// TIA Portal V18 export
FUNCTION_BLOCK "ST10_Flow2_A1TableUnloading"   // FB1072, GRAPH
// stored: AcknowledgeErrorsRequired false, AutoNumber false, GraphVersion 6.0, InitialValuesAcquisition false, SetENOAutomatically false
   // inherited from GRAPH_BASE
   VAR_INPUT
      iSysInface : "RCS_SysComInterface_V1";
   END_VAR
   VAR_IN_OUT
      ioPM_Inface : "RCS_PMInterface_V1";
      ioStatus : Int;
   END_VAR
   VAR
      sCtrlMode { S7_SetPoint := 'True'} : "SysFlowCtrlGraph";
      sUpdMES_Data : Bool;   // 更新MES数据
      工件放行中 : Bool;
      前站站号 { ExternalAccessible := 'False'; ExternalVisible := 'False'; ExternalWritable := 'False'} : UInt;
      本站站号 { ExternalAccessible := 'False'; ExternalVisible := 'False'; ExternalWritable := 'False'} : UInt;
      弹窗Temp : Array[1..10] of Int;
      AlarmID : Int;
      TON { S7_SetPoint := 'True'} : Array[0..10] of TON_TIME;
      TOF { S7_SetPoint := 'True'} : Array[0..10] of TOF_TIME;
      sUP { S7_SetPoint := 'True'} : Array[0..10] of Bool;
      更新RFID完成 : Bool;
   END_VAR
   VAR_TEMP
      Tempresult : USInt;
      本站站号乘10 : UInt;
   END_VAR
   // // TON[0] : 托盘流入1托盘到位传感器 / iA-Rotating product Check
   // // TON[1] : 托盘流入1托盘到位传感器
   // // TON[2] : 托盘流入1产品有无传感器
   // // TON[3] : 托盘流入1产品有无传感器
   // // TON[4] : 托盘流入1姿态检测光电2
   // // TON[5] : 托盘流入1姿态检测光电3
   // // TON[0].Q : 托盘流入1托盘到位 / iA-Rotating product Check
   // // TON[1].Q : 托盘流入1托盘无
   // // TON[2].Q : 托盘流入1有产品
   // // TON[3].Q : 托盘流入1无产品
   // // TON[4].Q : 托盘流入1姿态检测光电2
   // // TON[5].Q : 托盘流入1姿态检测光电3
   // // TOF[1] : iA-Rotating product Check
BEGIN
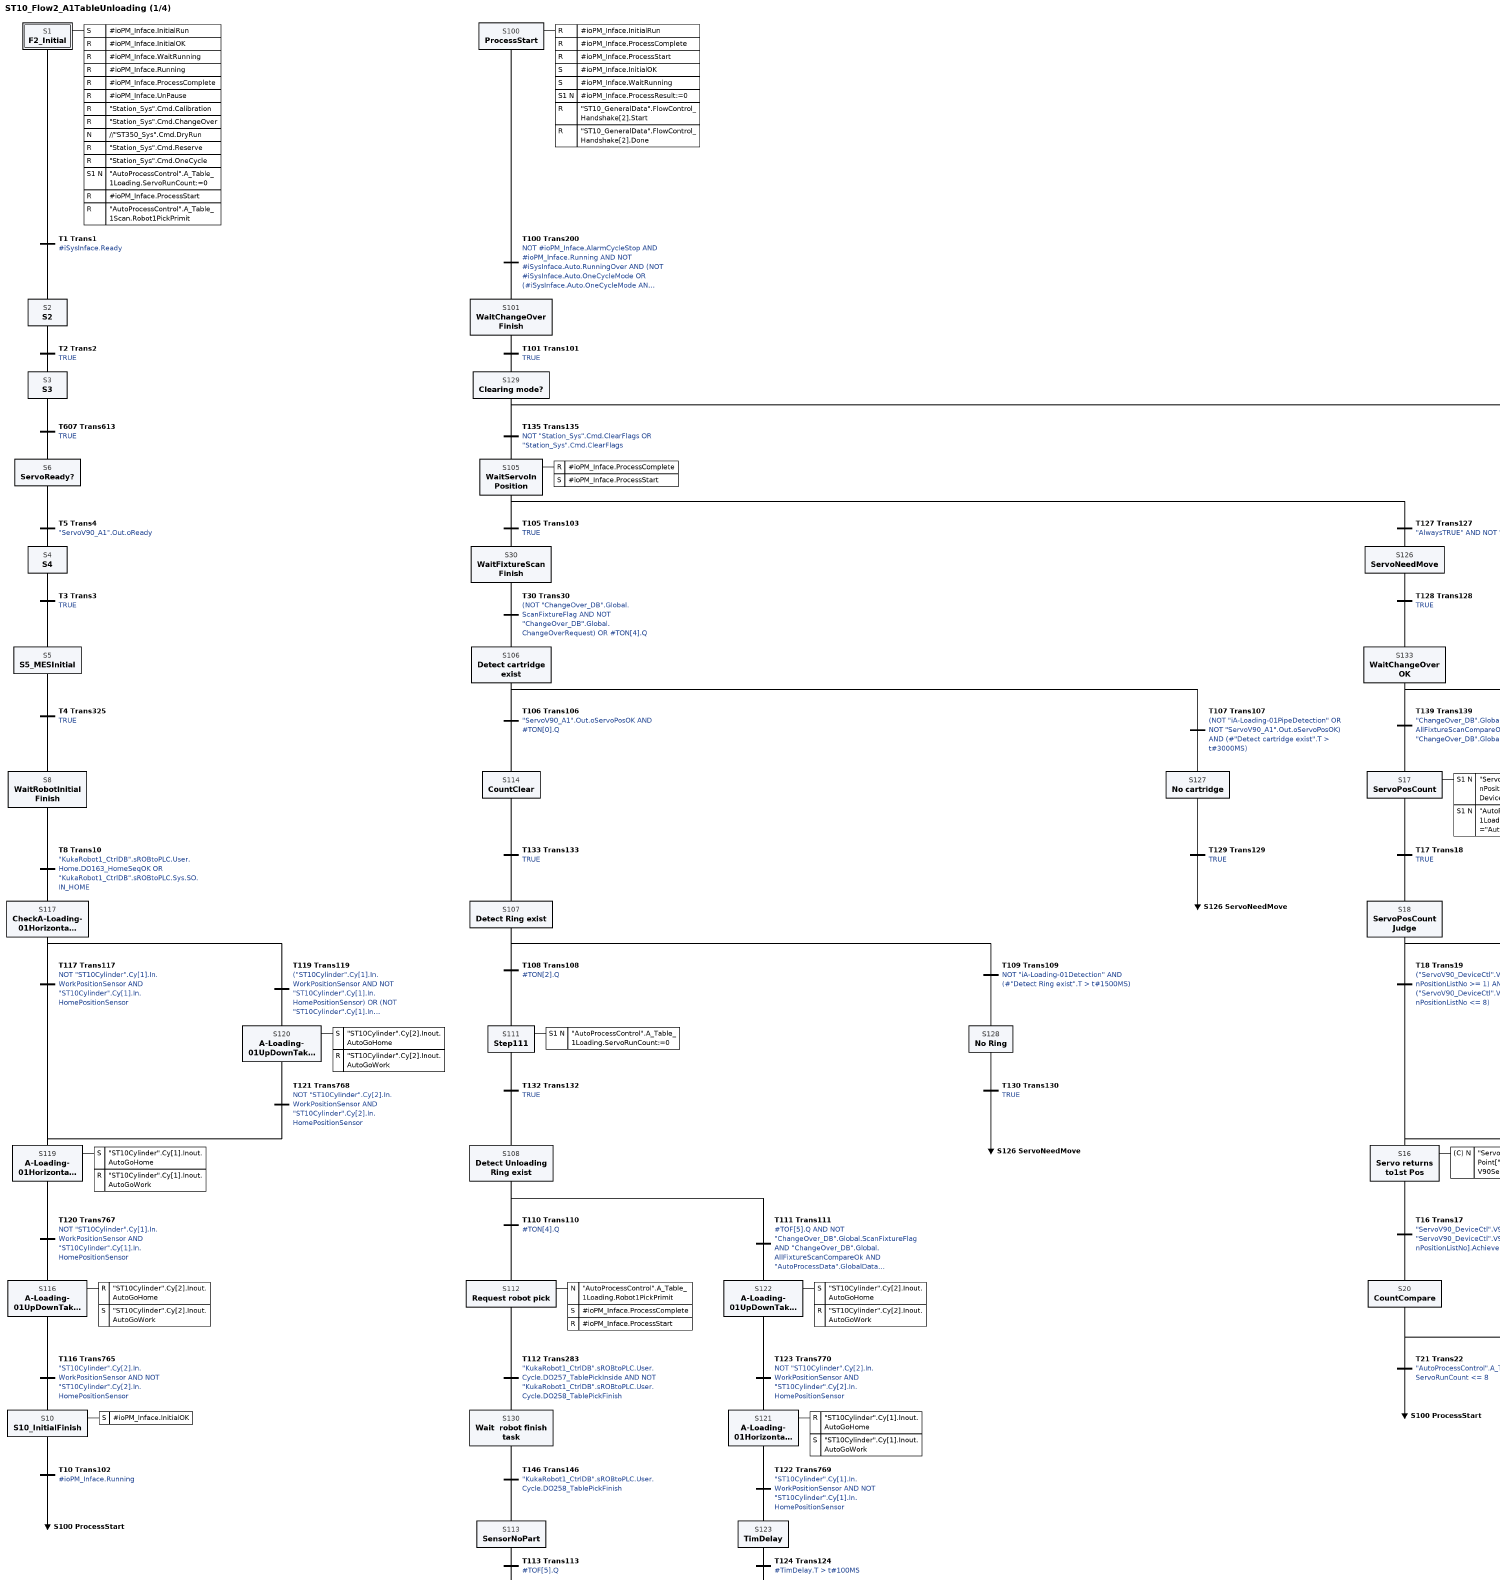
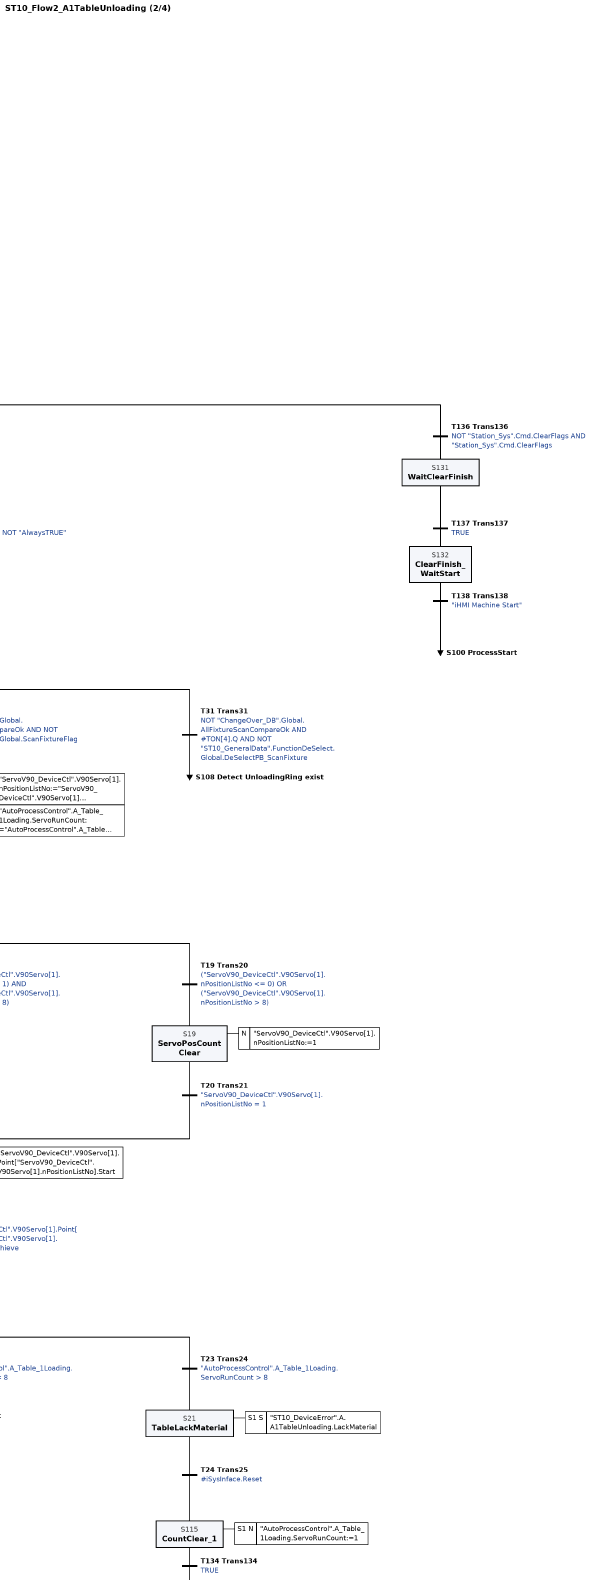
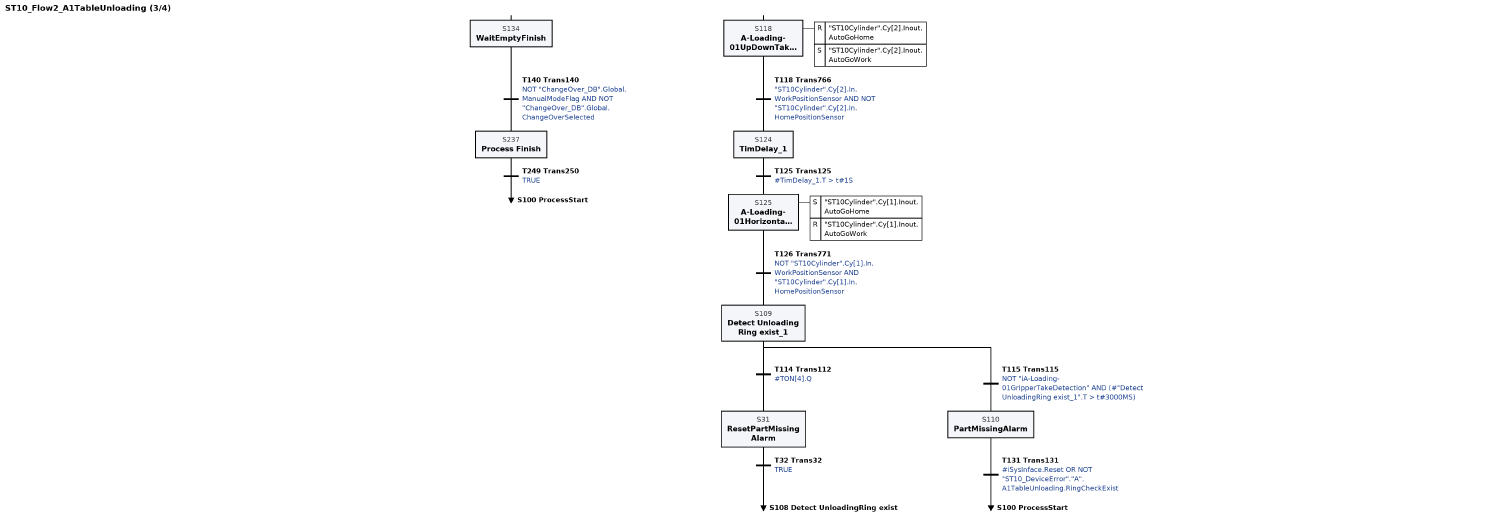
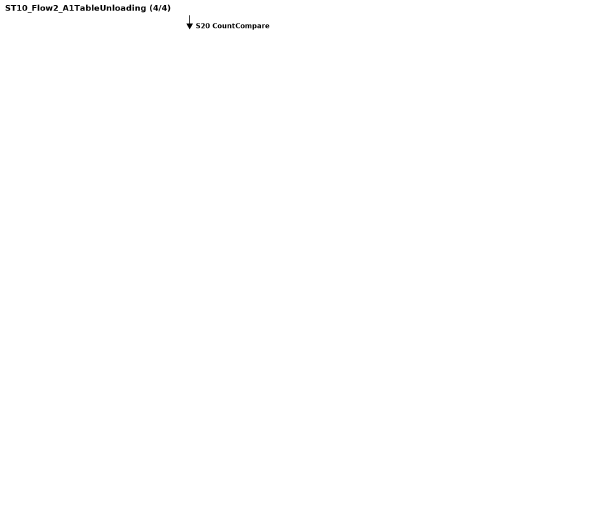
   // permanent pre-instructions
   NETWORK 1
      #TON[10].TON(IN := "AlwaysTRUE" AND "Station_Sys".Alarm.ImmediatelyStop, PT := T#300ms);
      #ioPM_Inface.AlarmImdilyStop := #TON[10].Q;
      #ioPM_Inface.AlarmCycleStop := "AlwaysTRUE" AND "Station_Sys".Alarm.CycleStop;
   NETWORK 2
      IF NOT False THEN
          #sCtrlMode(iSysInface := #iSysInface, ioPM_Inface := #ioPM_Inface, ioGraphCtrl := #RT_DATA.MOP);   // "SysFlowCtrlGraph"
      END_IF;
   NETWORK 3
      #TON[0].TON(IN := "AlwaysTRUE" AND "iA-Loading-01PipeDetection", PT := t#500ms);   // 工位11有托盘
      #TOF[1].TOF(IN := "AlwaysTRUE" AND NOT "iA-Loading-01PipeDetection", PT := T#300ms);   // 工位无托盘
      #TON[2].TON(IN := "AlwaysTRUE" AND "iA-Loading-01Detection", PT := T#300ms);
      #TOF[3].TOF(IN := "AlwaysTRUE" AND NOT "iA-Loading-01Detection", PT := T#300ms);
      #TON[4].TON(IN := "AlwaysTRUE" AND "iA-Loading-01GripperTakeDetection", PT := T#300ms);
      #TOF[5].TOF(IN := "AlwaysTRUE" AND NOT "iA-Loading-01GripperTakeDetection", PT := T#300ms);
   NETWORK 4
      #前站站号 := 345;
      #本站站号 := 350;

   // sequencer 1: S01-S99 初始化 / S01-S99 Initial
   INITIAL_STEP F2_Initial:   // S1, max time T#10S, warning time T#7S
              S    #ioPM_Inface.InitialRun
              R    #ioPM_Inface.InitialOK
              R    #ioPM_Inface.WaitRunning
              R    #ioPM_Inface.Running
              R    #ioPM_Inface.ProcessComplete
              R    #ioPM_Inface.UnPause
              R    "Station_Sys".Cmd.Calibration
              R    "Station_Sys".Cmd.ChangeOver
                   //"ST350_Sys".Cmd.DryRun
              R    "Station_Sys".Cmd.Reserve
              R    "Station_Sys".Cmd.OneCycle
          S1  N    "AutoProcessControl".A_Table_1Loading.ServoRunCount:=0
              R    #ioPM_Inface.ProcessStart
              R    "AutoProcessControl".A_Table_1Scan.Robot1PickPrimit
              R    "AutoProcessControl".A_Table_1Loading.Robot1PickPrimit
              R    "AutoProcessControl".A_Table_2Scan.Robot3PickPrimit
              R    "AutoProcessControl".A_Table_2Loading.Robot3PickPrimit
              R    "AutoProcessControl".A_ScanRotary.Robot1PickPrimit
              R    "AutoProcessControl".A_ScanRotary.Robot1PutPrimit
              R    "AutoProcessControl".H_ShafeLine.Robot1PickPrimit
              R    "AutoProcessControl".J_MagnetLine.Robot2PickPrimit
              R    "AutoProcessControl".K_ShafeLine.Robot2PickPrimit
              R    "AutoProcessControl".L_ShafeLine.Robot3PutPrimit
   END_STEP
   TRANSITION Trans1 FROM F2_Initial TO S2   // T1
      := #iSysInface.Ready;
   END_TRANSITION
   STEP S2:   // S2, max time T#10S, warning time T#7S
   END_STEP
   TRANSITION Trans2 FROM S2 TO S3   // T2
      := TRUE;
   END_TRANSITION
   STEP S4:   // S4, max time T#10S, warning time T#7S
   END_STEP
   TRANSITION Trans3 FROM S4 TO S5_MESInitial   // T3
      := TRUE;
   END_TRANSITION
   STEP S5_MESInitial:   // S5, max time T#10S, warning time T#7S
   END_STEP
   TRANSITION Trans325 FROM S5_MESInitial TO WaitRobotInitialFinish   // T4
      := TRUE;
   END_TRANSITION
   STEP S10_InitialFinish:   // S10, max time T#10S, warning time T#7S
              S    #ioPM_Inface.InitialOK
   END_STEP
   TRANSITION Trans102 FROM S10_InitialFinish TO ProcessStart   // T10, jump
      := #ioPM_Inface.Running;
   END_TRANSITION
   STEP S3:   // S3, max time T#10S, warning time T#7S
   END_STEP
   TRANSITION Trans613 FROM S3 TO "ServoReady?"   // T607
      := TRUE;
   END_TRANSITION
   STEP WaitRobotInitialFinish:   // S8, max time T#10S, warning time T#7S
   END_STEP
   TRANSITION Trans10 FROM WaitRobotInitialFinish TO "CheckA-Loading-01HorizontalCylindePos"   // T8
      := "KukaRobot1_CtrlDB".sROBtoPLC.User.Home.DO163_HomeSeqOK OR "KukaRobot1_CtrlDB".sROBtoPLC.Sys.SO.IN_HOME;
   END_TRANSITION
   STEP "A-Loading-01UpDownTakeCylinderToHP_2":   // S120, max time T#10S, warning time T#7S
              S    "ST10Cylinder".Cy[2].Inout.AutoGoHome
              R    "ST10Cylinder".Cy[2].Inout.AutoGoWork
   END_STEP
   TRANSITION Trans768 FROM "A-Loading-01UpDownTakeCylinderToHP_2" TO "A-Loading-01HorizontalCylinderToHP"   // T121
      := NOT "ST10Cylinder".Cy[2].In.WorkPositionSensor AND "ST10Cylinder".Cy[2].In.HomePositionSensor;
   END_TRANSITION
   STEP "CheckA-Loading-01HorizontalCylindePos":   // S117, max time T#10S, warning time T#7S
   END_STEP
   TRANSITION Trans117 FROM "CheckA-Loading-01HorizontalCylindePos" TO "A-Loading-01HorizontalCylinderToHP"   // T117
      := NOT "ST10Cylinder".Cy[1].In.WorkPositionSensor AND "ST10Cylinder".Cy[1].In.HomePositionSensor;
   END_TRANSITION
   TRANSITION Trans119 FROM "CheckA-Loading-01HorizontalCylindePos" TO "A-Loading-01UpDownTakeCylinderToHP_2"   // T119
      := ("ST10Cylinder".Cy[1].In.WorkPositionSensor AND NOT "ST10Cylinder".Cy[1].In.HomePositionSensor) OR (NOT "ST10Cylinder".Cy[1].In.WorkPositionSensor AND NOT "ST10Cylinder".Cy[1].In.HomePositionSensor);
   END_TRANSITION
   STEP "A-Loading-01HorizontalCylinderToHP":   // S119, max time T#10S, warning time T#7S
              S    "ST10Cylinder".Cy[1].Inout.AutoGoHome
              R    "ST10Cylinder".Cy[1].Inout.AutoGoWork
   END_STEP
   TRANSITION Trans767 FROM "A-Loading-01HorizontalCylinderToHP" TO "A-Loading-01UpDownTakeCylinderToWP"   // T120
      := NOT "ST10Cylinder".Cy[1].In.WorkPositionSensor AND "ST10Cylinder".Cy[1].In.HomePositionSensor;
   END_TRANSITION
   STEP "A-Loading-01UpDownTakeCylinderToWP":   // S116, max time T#10S, warning time T#7S
              R    "ST10Cylinder".Cy[2].Inout.AutoGoHome
              S    "ST10Cylinder".Cy[2].Inout.AutoGoWork
   END_STEP
   TRANSITION Trans765 FROM "A-Loading-01UpDownTakeCylinderToWP" TO S10_InitialFinish   // T116
      := "ST10Cylinder".Cy[2].In.WorkPositionSensor AND NOT "ST10Cylinder".Cy[2].In.HomePositionSensor;
   END_TRANSITION
   STEP "ServoReady?":   // S6, max time T#10S, warning time T#7S
   END_STEP
   TRANSITION Trans4 FROM "ServoReady?" TO S4   // T5
      := "ServoV90_A1".Out.oReady;
   END_TRANSITION

   // sequencer 2: S100-S199 等待到位 / S100-S199 CheckSysStatus
   STEP "A-Loading-01HorizontalCylinderToWP_1":   // S121, max time T#10S, warning time T#7S
              R    "ST10Cylinder".Cy[1].Inout.AutoGoHome
              S    "ST10Cylinder".Cy[1].Inout.AutoGoWork
   END_STEP
   TRANSITION Trans769 FROM "A-Loading-01HorizontalCylinderToWP_1" TO TimDelay   // T122
      := "ST10Cylinder".Cy[1].In.WorkPositionSensor AND NOT "ST10Cylinder".Cy[1].In.HomePositionSensor;
   END_TRANSITION
   STEP "A-Loading-01UpDownTakeCylinderToHP3":   // S122, max time T#10S, warning time T#7S
              S    "ST10Cylinder".Cy[2].Inout.AutoGoHome
              R    "ST10Cylinder".Cy[2].Inout.AutoGoWork
   END_STEP
   TRANSITION Trans770 FROM "A-Loading-01UpDownTakeCylinderToHP3" TO "A-Loading-01HorizontalCylinderToWP_1"   // T123
      := NOT "ST10Cylinder".Cy[2].In.WorkPositionSensor AND "ST10Cylinder".Cy[2].In.HomePositionSensor;
   END_TRANSITION
   STEP TimDelay:   // S123, max time T#10S, warning time T#7S
   END_STEP
   TRANSITION Trans124 FROM TimDelay TO "A-Loading-01UpDownTakeCylinderToWP_1"   // T124
      := #TimDelay.T > t#100MS;
   END_TRANSITION
   STEP SensorNoPart:   // S113, max time T#10S, warning time T#7S
   END_STEP
   TRANSITION Trans113 FROM SensorNoPart TO WaitEmptyFinish   // T113
      := #TOF[5].Q;
   END_TRANSITION
   STEP ProcessStart:   // S100, max time T#10S, warning time T#7S
      // 自动等待开始运行
              R    #ioPM_Inface.InitialRun
              R    #ioPM_Inface.ProcessComplete
              R    #ioPM_Inface.ProcessStart
              S    #ioPM_Inface.InitialOK
              S    #ioPM_Inface.WaitRunning
          S1  N    #ioPM_Inface.ProcessResult:=0
              R    "ST10_GeneralData".FlowControl_Handshake[2].Start
              R    "ST10_GeneralData".FlowControl_Handshake[2].Done
   END_STEP
   TRANSITION Trans200 FROM ProcessStart TO WaitChangeOverFinish   // T100
      := NOT #ioPM_Inface.AlarmCycleStop AND #ioPM_Inface.Running AND NOT #iSysInface.Auto.RunningOver AND (NOT #iSysInface.Auto.OneCycleMode OR (#iSysInface.Auto.OneCycleMode AND #ioPM_Inface.TriggerOneCycle));
   END_TRANSITION
   STEP TimDelay_1:   // S124, max time T#10S, warning time T#7S
   END_STEP
   TRANSITION Trans125 FROM TimDelay_1 TO "A-Loading-01HorizontalCylinderToHP_1"   // T125
      := #TimDelay_1.T > t#1S;
   END_TRANSITION
   STEP "Process Finish":   // S237, max time T#10S, warning time T#7S
   END_STEP
   TRANSITION Trans250 FROM "Process Finish" TO ProcessStart   // T249, jump
      := TRUE;
   END_TRANSITION
   STEP "A-Loading-01HorizontalCylinderToHP_1":   // S125, max time T#10S, warning time T#7S
              S    "ST10Cylinder".Cy[1].Inout.AutoGoHome
              R    "ST10Cylinder".Cy[1].Inout.AutoGoWork
   END_STEP
   TRANSITION Trans771 FROM "A-Loading-01HorizontalCylinderToHP_1" TO "Detect UnloadingRing exist_1"   // T126
      := NOT "ST10Cylinder".Cy[1].In.WorkPositionSensor AND "ST10Cylinder".Cy[1].In.HomePositionSensor;
   END_TRANSITION
   STEP "No cartridge":   // S127, max time T#10S, warning time T#7S
   END_STEP
   TRANSITION Trans129 FROM "No cartridge" TO ServoNeedMove   // T129, jump
      := TRUE;
   END_TRANSITION
   STEP "A-Loading-01UpDownTakeCylinderToWP_1":   // S118, max time T#10S, warning time T#7S
              R    "ST10Cylinder".Cy[2].Inout.AutoGoHome
              S    "ST10Cylinder".Cy[2].Inout.AutoGoWork
   END_STEP
   TRANSITION Trans766 FROM "A-Loading-01UpDownTakeCylinderToWP_1" TO TimDelay_1   // T118
      := "ST10Cylinder".Cy[2].In.WorkPositionSensor AND NOT "ST10Cylinder".Cy[2].In.HomePositionSensor;
   END_TRANSITION
   STEP ServoNeedMove:   // S126, max time T#10S, warning time T#7S
   END_STEP
   TRANSITION Trans128 FROM ServoNeedMove TO WaitChangeOverOK   // T128
      := TRUE;
   END_TRANSITION
   STEP WaitChangeOverFinish:   // S101, max time T#10S, warning time T#7S
   END_STEP
   TRANSITION Trans101 FROM WaitChangeOverFinish TO "Clearing mode?"   // T101
      := TRUE;
   END_TRANSITION
   STEP WaitServoInPosition:   // S105, max time T#10S, warning time T#7S
              R    #ioPM_Inface.ProcessComplete
              S    #ioPM_Inface.ProcessStart
   END_STEP
   TRANSITION Trans103 FROM WaitServoInPosition TO WaitFixtureScanFinish   // T105
      := TRUE;
   END_TRANSITION
   TRANSITION Trans127 FROM WaitServoInPosition TO ServoNeedMove   // T127
      := "AlwaysTRUE" AND NOT "AlwaysTRUE";
   END_TRANSITION
   STEP "Detect cartridge exist":   // S106, max time T#10S, warning time T#7S
   END_STEP
   TRANSITION Trans106 FROM "Detect cartridge exist" TO CountClear   // T106
      := "ServoV90_A1".Out.oServoPosOK AND #TON[0].Q;
   END_TRANSITION
   TRANSITION Trans107 FROM "Detect cartridge exist" TO "No cartridge"   // T107
      := (NOT "iA-Loading-01PipeDetection" OR NOT "ServoV90_A1".Out.oServoPosOK) AND (#"Detect cartridge exist".T > t#3000MS);
   END_TRANSITION
   STEP "Detect UnloadingRing exist":   // S108, max time T#10S, warning time T#7S
   END_STEP
   TRANSITION Trans110 FROM "Detect UnloadingRing exist" TO "Request robot pick"   // T110
      := #TON[4].Q;
   END_TRANSITION
   TRANSITION Trans111 FROM "Detect UnloadingRing exist" TO "A-Loading-01UpDownTakeCylinderToHP3"   // T111
      := #TOF[5].Q AND NOT "ChangeOver_DB".Global.ScanFixtureFlag AND "ChangeOver_DB".Global.AllFixtureScanCompareOk AND "AutoProcessData".GlobalData.Table1CodeOKFlag;
   END_TRANSITION
   STEP "Detect Ring exist":   // S107, max time T#10S, warning time T#7S
   END_STEP
   TRANSITION Trans108 FROM "Detect Ring exist" TO Step111   // T108
      := #TON[2].Q;
   END_TRANSITION
   TRANSITION Trans109 FROM "Detect Ring exist" TO "No Ring"   // T109
      := NOT "iA-Loading-01Detection" AND (#"Detect Ring exist".T > t#1500MS);
   END_TRANSITION
   STEP "Wait  robot finish task":   // S130, max time T#10S, warning time T#7S
   END_STEP
   TRANSITION Trans146 FROM "Wait  robot finish task" TO SensorNoPart   // T146
      := "KukaRobot1_CtrlDB".sROBtoPLC.User.Cycle.DO258_TablePickFinish;
   END_TRANSITION
   STEP "Request robot pick":   // S112, max time T#10S, warning time T#7S
              N    "AutoProcessControl".A_Table_1Loading.Robot1PickPrimit
              S    #ioPM_Inface.ProcessComplete
              R    #ioPM_Inface.ProcessStart
   END_STEP
   TRANSITION Trans283 FROM "Request robot pick" TO "Wait  robot finish task"   // T112
      := "KukaRobot1_CtrlDB".sROBtoPLC.User.Cycle.DO257_TablePickInside AND NOT "KukaRobot1_CtrlDB".sROBtoPLC.User.Cycle.DO258_TablePickFinish;
   END_TRANSITION
   STEP "No Ring":   // S128, max time T#10S, warning time T#7S
   END_STEP
   TRANSITION Trans130 FROM "No Ring" TO ServoNeedMove   // T130, jump
      := TRUE;
   END_TRANSITION
   STEP "Detect UnloadingRing exist_1":   // S109, max time T#10S, warning time T#7S
   END_STEP
   TRANSITION Trans112 FROM "Detect UnloadingRing exist_1" TO ResetPartMissingAlarm   // T114
      := #TON[4].Q;
   END_TRANSITION
   TRANSITION Trans115 FROM "Detect UnloadingRing exist_1" TO PartMissingAlarm   // T115
      := NOT "iA-Loading-01GripperTakeDetection" AND (#"Detect UnloadingRing exist_1".T > t#3000MS);
   END_TRANSITION
   STEP PartMissingAlarm:   // S110, max time T#10S, warning time T#7S
   END_STEP
   TRANSITION Trans131 FROM PartMissingAlarm TO ProcessStart   // T131, jump
      := #iSysInface.Reset OR NOT "ST10_DeviceError"."A".A1TableUnloading.RingCheckExist;
   END_TRANSITION
   STEP Step111:   // S111, max time T#10S, warning time T#7S
          S1  N    "AutoProcessControl".A_Table_1Loading.ServoRunCount:=0
   END_STEP
   TRANSITION Trans132 FROM Step111 TO "Detect UnloadingRing exist"   // T132
      := TRUE;
   END_TRANSITION
   STEP CountClear:   // S114, max time T#10S, warning time T#7S
   END_STEP
   TRANSITION Trans133 FROM CountClear TO "Detect Ring exist"   // T133
      := TRUE;
   END_TRANSITION
   STEP "Servo returns to1st Pos":   // S16, max time T#10S, warning time T#7S
      interlock C := "ServoV90_A1".Out.oReady;
      (C)     N    "ServoV90_DeviceCtl".V90Servo[1].Point["ServoV90_DeviceCtl".V90Servo[1].nPositionListNo].Start
   END_STEP
   TRANSITION Trans17 FROM "Servo returns to1st Pos" TO CountCompare   // T16
      := "ServoV90_DeviceCtl".V90Servo[1].Point["ServoV90_DeviceCtl".V90Servo[1].nPositionListNo].Achieve;
   END_TRANSITION
   STEP ServoPosCount:   // S17, max time T#10S, warning time T#7S
          S1  N    "ServoV90_DeviceCtl".V90Servo[1].nPositionListNo:="ServoV90_DeviceCtl".V90Servo[1].nPositionListNo+1
          S1  N    "AutoProcessControl".A_Table_1Loading.ServoRunCount:="AutoProcessControl".A_Table_1Loading.ServoRunCount+1
   END_STEP
   TRANSITION Trans18 FROM ServoPosCount TO ServoPosCountJudge   // T17
      := TRUE;
   END_TRANSITION
   STEP ServoPosCountJudge:   // S18, max time T#10S, warning time T#7S
   END_STEP
   TRANSITION Trans19 FROM ServoPosCountJudge TO "Servo returns to1st Pos"   // T18
      := ("ServoV90_DeviceCtl".V90Servo[1].nPositionListNo >= 1) AND ("ServoV90_DeviceCtl".V90Servo[1].nPositionListNo <= 8);
   END_TRANSITION
   TRANSITION Trans20 FROM ServoPosCountJudge TO ServoPosCountClear   // T19
      := ("ServoV90_DeviceCtl".V90Servo[1].nPositionListNo <= 0) OR ("ServoV90_DeviceCtl".V90Servo[1].nPositionListNo > 8);
   END_TRANSITION
   STEP ServoPosCountClear:   // S19, max time T#10S, warning time T#7S
              N    "ServoV90_DeviceCtl".V90Servo[1].nPositionListNo:=1
   END_STEP
   TRANSITION Trans21 FROM ServoPosCountClear TO "Servo returns to1st Pos"   // T20
      := "ServoV90_DeviceCtl".V90Servo[1].nPositionListNo = 1;
   END_TRANSITION
   STEP CountCompare:   // S20, max time T#10S, warning time T#7S
   END_STEP
   TRANSITION Trans22 FROM CountCompare TO ProcessStart   // T21, jump
      := "AutoProcessControl".A_Table_1Loading.ServoRunCount <= 8;
   END_TRANSITION
   TRANSITION Trans24 FROM CountCompare TO TableLackMaterial   // T23
      := "AutoProcessControl".A_Table_1Loading.ServoRunCount > 8;
   END_TRANSITION
   STEP TableLackMaterial:   // S21, max time T#10S, warning time T#7S
          S1  S    "ST10_DeviceError".A.A1TableUnloading.LackMaterial
   END_STEP
   TRANSITION Trans25 FROM TableLackMaterial TO CountClear_1   // T24
      := #iSysInface.Reset;
   END_TRANSITION
   STEP CountClear_1:   // S115, max time T#10S, warning time T#7S
          S1  N    "AutoProcessControl".A_Table_1Loading.ServoRunCount:=1
   END_STEP
   TRANSITION Trans134 FROM CountClear_1 TO CountCompare   // T134, jump
      := TRUE;
   END_TRANSITION
   STEP "Clearing mode?":   // S129, max time T#10S, warning time T#7S
   END_STEP
   TRANSITION Trans135 FROM "Clearing mode?" TO WaitServoInPosition   // T135
      := NOT "Station_Sys".Cmd.ClearFlags OR "Station_Sys".Cmd.ClearFlags;
   END_TRANSITION
   TRANSITION Trans136 FROM "Clearing mode?" TO WaitClearFinish   // T136
      := NOT "Station_Sys".Cmd.ClearFlags AND "Station_Sys".Cmd.ClearFlags;
   END_TRANSITION
   STEP WaitClearFinish:   // S131, max time T#10S, warning time T#7S
   END_STEP
   TRANSITION Trans137 FROM WaitClearFinish TO ClearFinish_WaitStart   // T137
      := TRUE;
   END_TRANSITION
   STEP ClearFinish_WaitStart:   // S132, max time T#10S, warning time T#7S
   END_STEP
   TRANSITION Trans138 FROM ClearFinish_WaitStart TO ProcessStart   // T138, jump
      := "iHMI Machine Start";
   END_TRANSITION
   STEP WaitChangeOverOK:   // S133, max time T#10S, warning time T#7S
   END_STEP
   TRANSITION Trans139 FROM WaitChangeOverOK TO ServoPosCount   // T139
      := "ChangeOver_DB".Global.AllFixtureScanCompareOk AND NOT "ChangeOver_DB".Global.ScanFixtureFlag;
   END_TRANSITION
   TRANSITION Trans31 FROM WaitChangeOverOK TO "Detect UnloadingRing exist"   // T31, jump
      := NOT "ChangeOver_DB".Global.AllFixtureScanCompareOk AND #TON[4].Q AND NOT "ST10_GeneralData".FunctionDeSelect.Global.DeSelectPB_ScanFixture;
   END_TRANSITION
   STEP WaitEmptyFinish:   // S134, max time T#10S, warning time T#7S
   END_STEP
   TRANSITION Trans140 FROM WaitEmptyFinish TO "Process Finish"   // T140
      := NOT "ChangeOver_DB".Global.ManualModeFlag AND NOT "ChangeOver_DB".Global.ChangeOverSelected;
   END_TRANSITION
   STEP WaitFixtureScanFinish:   // S30, max time T#10S, warning time T#7S
   END_STEP
   TRANSITION Trans30 FROM WaitFixtureScanFinish TO "Detect cartridge exist"   // T30
      := (NOT "ChangeOver_DB".Global.ScanFixtureFlag AND NOT "ChangeOver_DB".Global.ChangeOverRequest) OR #TON[4].Q;
   END_TRANSITION
   STEP ResetPartMissingAlarm:   // S31, max time T#10S, warning time T#7S
   END_STEP
   TRANSITION Trans32 FROM ResetPartMissingAlarm TO "Detect UnloadingRing exist"   // T32, jump
      := TRUE;
   END_TRANSITION

   // permanent post-instructions
   NETWORK 1
      #ioPM_Inface.StepNum := #RT_DATA.S_DISPLAY;
   NETWORK 2
      IF #iSysInface.Reset THEN #AlarmID := 0; END_IF;
   NETWORK 3
      #TON[10].TON(IN := #工件放行中, PT := T#0.5S);
      IF #TON[10].Q THEN #工件放行中 := FALSE; END_IF;
END_FUNCTION_BLOCK
